TEXTLIST Mc_Warnings
  0 = 'Machine Warning 0'
  1 = 'Warning 2'
  2 = 'Warning 3'
  3 = 'Low Oil Level'
   = ''
END_TEXTLIST

(* stored: Version 1.1.0.1, ProductVersion 3.1.4024.12
   TextList Mc_Warnings: Id {fd185ce1-9315-01c5-104f-3e9e22efccb8} *)
